FUNCTION_BLOCK FB_System_BelHa_Ablaufsteuerung
VAR_IN_OUT
	Zustand			: ST_System_Bel_Zustand;
	Stellwert		: ST_System_Bel_Stellwert;
END_VAR
VAR_INPUT
	Steuerung		: ST_System_Bel_Steuerung;
	Parameter		: ST_System_Bel_Parameter;
END_VAR
VAR_OUTPUT
END_VAR
VAR
	Timer: TON;
END_VAR

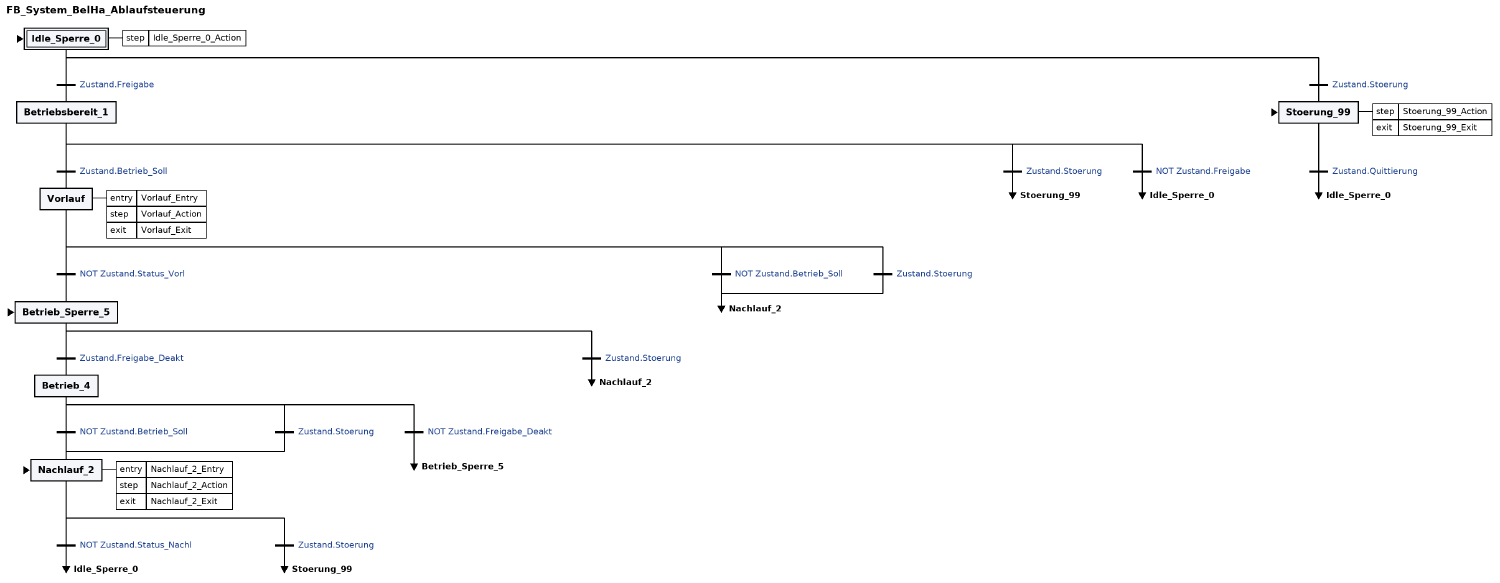
INITIAL_STEP Idle_Sperre_0:
    Idle_Sperre_0_Action(N);  // step action
END_STEP
TRANSITION FROM Idle_Sperre_0 TO Betriebsbereit_1
    := Zustand.Freigabe;
END_TRANSITION
TRANSITION FROM Idle_Sperre_0 TO Stoerung_99
    := Zustand.Stoerung;
END_TRANSITION
STEP Stoerung_99:
    Stoerung_99_Action(N);  // step action
    Stoerung_99_Exit(P0);  // exit action
END_STEP
TRANSITION FROM Stoerung_99 TO Idle_Sperre_0
    := Zustand.Quittierung;
END_TRANSITION
STEP Betriebsbereit_1:
END_STEP
TRANSITION FROM Betriebsbereit_1 TO Vorlauf
    := Zustand.Betrieb_Soll;
END_TRANSITION
TRANSITION FROM Betriebsbereit_1 TO Stoerung_99
    := Zustand.Stoerung;
END_TRANSITION
TRANSITION FROM Betriebsbereit_1 TO Idle_Sperre_0
    := NOT Zustand.Freigabe;
END_TRANSITION
STEP Vorlauf:
    Vorlauf_Entry(P1);  // entry action
    Vorlauf_Action(N);  // step action
    Vorlauf_Exit(P0);  // exit action
END_STEP
TRANSITION FROM Vorlauf TO Betrieb_Sperre_5
    := NOT Zustand.Status_Vorl;
END_TRANSITION
TRANSITION FROM Vorlauf TO Nachlauf_2
    := NOT Zustand.Betrieb_Soll;
END_TRANSITION
TRANSITION FROM Vorlauf TO Nachlauf_2
    := Zustand.Stoerung;
END_TRANSITION
STEP Betrieb_Sperre_5:
END_STEP
TRANSITION FROM Betrieb_Sperre_5 TO Betrieb_4
    := Zustand.Freigabe_Deakt;
END_TRANSITION
TRANSITION FROM Betrieb_Sperre_5 TO Nachlauf_2
    := Zustand.Stoerung;
END_TRANSITION
STEP Betrieb_4:
END_STEP
TRANSITION FROM Betrieb_4 TO Nachlauf_2
    := NOT Zustand.Betrieb_Soll;
END_TRANSITION
TRANSITION FROM Betrieb_4 TO Nachlauf_2
    := Zustand.Stoerung;
END_TRANSITION
TRANSITION FROM Betrieb_4 TO Betrieb_Sperre_5
    := NOT Zustand.Freigabe_Deakt;
END_TRANSITION
STEP Nachlauf_2:
    Nachlauf_2_Entry(P1);  // entry action
    Nachlauf_2_Action(N);  // step action
    Nachlauf_2_Exit(P0);  // exit action
END_STEP
TRANSITION FROM Nachlauf_2 TO Idle_Sperre_0
    := NOT Zustand.Status_Nachl;
END_TRANSITION
TRANSITION FROM Nachlauf_2 TO Stoerung_99
    := Zustand.Stoerung;
END_TRANSITION

ACTION Idle_Sperre_0_Action:
(* Quittierungszustand auf False setzen, damit das System bei einer erneuten Störung nicht direkt wieder angeschaltet wird *)
Steuerung.Quittierung	:= FALSE;
END_ACTION

ACTION Nachlauf_2_Action:
(* Nachlauf Timer starten *)
Timer( 	IN := Zustand.Status_Nachl,
		PT := DINT_TO_TIME(Parameter.Zeit_Nachl)
);
Zustand.Status_Nachl	:= NOT(Timer.Q AND NOT Zustand.Betrieb);

(* Stellwert setzen *)
Stellwert.Betrieb := FALSE;

(* Zustand setzen *)
Zustand.Status := E_Bel_Zustand_Status_Nachl;
END_ACTION

ACTION Nachlauf_2_Entry:
Zustand.Status_Nachl := TRUE;
(* Reset Timer *)
Timer(IN := FALSE);
END_ACTION

ACTION Nachlauf_2_Exit:
Zustand.Status_Nachl := FALSE;
END_ACTION

ACTION Stoerung_99_Action:
(* Stellwert setzen *)
Stellwert.Betrieb := FALSE;

(* Zustand setzen *)
Zustand.Stoerung := TRUE;
Zustand.Status := E_Bel_Zustand_Status_Stoerung;
END_ACTION

ACTION Stoerung_99_Exit:
Zustand.Stoerung	:= FALSE;
END_ACTION

ACTION Vorlauf_Action:
(* Vorlaufzeit Timer starten *)
Timer( 	IN := Zustand.Status_Vorl,
		PT := DINT_TO_TIME(Parameter.Zeit_Vorl)
);
Zustand.Status_Vorl := NOT (Timer.Q AND Zustand.Betrieb);

(* Stellwert setzen *)
Stellwert.Betrieb 	:= TRUE;
Stellwert.Leistung  := Zustand.Leistung;
(* Zustand setzen *)
Zustand.Status := E_Bel_Zustand_Status_Vorl;
END_ACTION

ACTION Vorlauf_Entry:
Zustand.Status_Vorl := TRUE;
(* Reset Timer *)
Timer(IN := FALSE);
END_ACTION

ACTION Vorlauf_Exit:
Zustand.Status_Vorl := FALSE;
END_ACTION

END_FUNCTION_BLOCK

(* stored: Version 1.1.0.1, ProductVersion 3.1.4024.9
   POU FB_System_BelHa_Ablaufsteuerung: Id {99ce0e58-e3a0-4255-a411-257e6dc6adb2}, SpecialFunc None
   Action Idle_Sperre_0_Action: Id {e985e4e7-7c5e-4ae8-ae82-e38f9295037e}
   Action Nachlauf_2_Action: Id {b5683402-79ee-4b91-b076-78146681904a}
   Action Nachlauf_2_Entry: Id {2ee8d7be-a007-4892-ac69-0a520efa168d}
   Action Nachlauf_2_Exit: Id {c02597c3-a414-4349-9b5a-87581d4aac1e}
   Action Stoerung_99_Action: Id {fba42a6f-0dc1-40db-b022-b02a1aa10203}
   Action Stoerung_99_Exit: Id {6a16b667-bc94-4cf9-a688-1090e53da945}
   Action Vorlauf_Action: Id {0fd7a26a-98cd-4eec-8e57-4dbf6c1c0a8a}
   Action Vorlauf_Entry: Id {86067ae3-3b40-4e46-a5af-5e53d66c6f4d}
   Action Vorlauf_Exit: Id {736598fa-3b41-4940-b520-c57cf10e53e9} *)
